// TIA Portal V17 export
// export: Created 2024-09-02T12:50:33.2610661Z, ExportSetting WithDefaults, DisplayName Totally Integrated Automation Portal, DisplayVersion V17, DisplayName TIA Portal Openness, DisplayVersion V17, DisplayName TIA Portal Version Control Interface, DisplayVersion V17, DisplayName STEP 7 Professional, DisplayVersion V17, DisplayName STEP 7 Safety, DisplayVersion V17, DisplayName WinCC Professional, DisplayVersion V17
TYPE "TypeMobyHMIDiag"
// stored: IsFailsafeCompliant false
   STRUCT
      Done : Bool;   // Befehl wurde fehlerfrei ausgeführt / Command was executed without errors
      Busy : Bool;   // Der Baustein bearbeitet einen Befehl / The block processes a command
      Warning : Bool;   // Warnung wurde erkannt / Warning was detected
      Error : Bool;   // Fehler wurde erkannt / Error was detected
      Status : DWord;   // Warnung- und Fehler / Warning and error
      TransponderPresence : Bool;   // Transponder Presence
      TransponderPresenceChanged : Bool;   // Transponder Presence Changed
      iidCMDStruct { S7_SetPoint := 'True'} : IID_CMD_STRUCT;
   END_STRUCT;
END_TYPE
